{attribute 'qualified_only'}
{attribute 'strict'}
TYPE GripperCmd :
(
	noGrip := 0,
	take,
	put
);
END_TYPE

(* stored: Version 1.1.0.1, ProductVersion 3.1.4024.11
   DUT GripperCmd: Id {b80938dc-b405-4653-b69c-ada346329828} *)
